# EPICS substitutions: iocBoot/iocTest/testISIS_single.substitutions
file "db/testISIS.template" { pattern
{P, R, PORT, POLLER, INDEX, SLICE}
{omronEIP:, 0:, omronDriver, slowPoller, 1, 1}
{omronEIP:, 1:, omronDriver, slowPoller, 10, 1}
{omronEIP:, 2:, omronDriver, slowPoller, 19, 1}
{omronEIP:, 3:, omronDriver, slowPoller, 28, 1}
{omronEIP:, 4:, omronDriver, slowPoller, 37, 1}
{omronEIP:, 5:, omronDriver, fastPoller, 46, 1}
{omronEIP:, 6:, omronDriver, slowPoller, 55, 1}
}
